FUNCTION_BLOCK TcoTaskPlcTestObject EXTENDS TcoCore.TcoObject
VAR
    _myIdentity : ULINT;
    _myContextIdentity : ULINT;
    _myContextStartCount : ULINT;
    _myContextEndCount : ULINT;
    _myParentIdentity : ULINT;
    _sut_A : TcoTaskPlcTest(THIS^);
    _sut_B : TcoTaskPlcTest(THIS^);
    _tSt_A : TcoTaskPlcTestState(THIS^, eRestoreMode.AutoRestoreMembers);
    _tSt_B : TcoTaskPlcTestState(THIS^, eRestoreMode.None);
END_VAR

_sut_A();
_sut_B();

PROPERTY CounterValue_A : ULINT
GET
CounterValue_A := _sut_A.CounterValue;
END_GET
SET
_sut_A.CounterValue := CounterValue_A;
END_SET
END_PROPERTY

PROPERTY CounterValue_B : ULINT
GET
CounterValue_B := _sut_B.CounterValue;
END_GET
SET
_sut_B.CounterValue := CounterValue_B;
END_SET
END_PROPERTY

{attribute 'TcRpcEnable'}
METHOD INTERNAL ReadOutIdentities
_myIdentity := THIS^.Identity;
_myContextIdentity := THIS^.Context.Identity;
_myContextStartCount := THIS^.Context.StartCycleCount;
_myContextEndCount := THIS^.Context.EndCycleCount;
_myParentIdentity := THIS^.Parent.Identity;
END_METHOD

END_FUNCTION_BLOCK

(* stored: Version 1.1.0.1
   POU TcoTaskPlcTestObject: Id {e5a083e5-83f5-09f3-0c5b-570a13d7234f}, SpecialFunc None
   Property CounterValue_A: Id {5108df5b-bacd-0032-225a-5dc28c7c10cb}
   Get Get: Id {4023e99e-a54f-0fc9-0f5c-0c4e68f62e7c}
   Set Set: Id {4f0cf991-1e06-09c6-24ec-6f9fd9e46e40}
   Property CounterValue_B: Id {bd90ed58-5558-0599-29f7-42c0fd95ee77}
   Get Get: Id {883f80b3-84aa-06e3-2f8d-184bffe68342}
   Set Set: Id {9ce79a97-64cd-0048-15b6-fcc5d54125c9}
   Method ReadOutIdentities: Id {83ee5bb6-dfd6-0470-1384-2995dc5dc5b1} *)
